# EPICS IOC start-up script: examples/test/PSI/LLRF_ILK/v1/ILK.iocsh
#- #############################################################################
#- mXsXXX naming
require ecmccfg ILK_slaves, "ECMC_VER=dev,NAMING=mXsXXX"

#- add slaves
${SCRIPTEXEC} ${ecmccfg_DIR}addSlave.cmd, "HW_DESC=TOBAS"
${SCRIPTEXEC} ${ecmccfg_DIR}addSlave.cmd, "HW_DESC=EK1100"
${SCRIPTEXEC} ${ecmccfg_DIR}addSlave.cmd, "HW_DESC=EL1034"
${SCRIPTEXEC} ${ecmccfg_DIR}addSlave.cmd, "HW_DESC=EL1034"
${SCRIPTEXEC} ${ecmccfg_DIR}addSlave.cmd, "HW_DESC=EL1034"
${SCRIPTEXEC} ${ecmccfg_DIR}addSlave.cmd, "HW_DESC=EL1034"
${SCRIPTEXEC} ${ecmccfg_DIR}addSlave.cmd, "HW_DESC=EL1034"
${SCRIPTEXEC} ${ecmccfg_DIR}addSlave.cmd, "HW_DESC=EL2808"
${SCRIPTEXEC} ${ecmccfg_DIR}addSlave.cmd, "HW_DESC=EL3154"
${SCRIPTEXEC} ${ecmccfg_DIR}addSlave.cmd, "HW_DESC=EL3164"
${SCRIPTEXEC} ${ecmccfg_DIR}addSlave.cmd, "HW_DESC=EL1862"
${SCRIPTEXEC} ${ecmccfg_DIR}addSlave.cmd, "HW_DESC=EL1862"
${SCRIPTEXEC} ${ecmccfg_DIR}addSlave.cmd, "HW_DESC=ILK"

#- PLC for slave to slave bit transfer
$(SCRIPTEXEC) $(ecmccfg_DIR)loadPLCFile.cmd, "PLC_ID=0, SAMPLE_RATE_MS=1,FILE=./plc/ena.plc")
